FUNCTION_BLOCK FB_Crane
VAR_INPUT
END_VAR
VAR_OUTPUT
END_VAR
VAR
END_VAR

END_FUNCTION_BLOCK

(* stored: Version 1.1.0.1, ProductVersion 3.1.4024.16
   POU FB_Crane: Id {b92e7889-f852-4a96-a33c-3002a177f6c5}, SpecialFunc None *)
